Fanuc KAREL source: inv_sys.kl

PROGRAM INV_SYS
%SYSTEM
%INVISIBLE
VAR
	I : INTEGER
BEGIN
	I = 1
	WRITE('I = ', I, CR)
END INV_SYS
